// TIA Portal V17 export
// export: Created 2022-07-28T18:02:49.3810425Z, ExportSetting None, DisplayName Totally Integrated Automation Portal, DisplayVersion V17, DisplayName TIA Portal Openness, DisplayVersion V17, DisplayName TIA Portal Teamcenter Gateway, DisplayVersion V17, DisplayName TIA Portal Version Control Interface, DisplayVersion V17, DisplayName TIA Portal Test Suite Advanced, DisplayVersion V17, DisplayName SINAMICS Startdrive Advanced, DisplayVersion V17, DisplayName SINAMICS DCC, DisplayVersion V17, DisplayName SINAMICS Startdrive G130, G150, S120, S150, SINAMICS MV, S210, DisplayVersion V17, DisplayName SINAMICS Startdrive G110M, G120, G120C, G120D, G120P, G115D, DisplayVersion V17, DisplayName STEP 7 Professional, DisplayVersion V17, DisplayName SIMATIC Energy Suite, DisplayVersion V17, DisplayName STEP 7 CFC, DisplayVersion V17, DisplayName STEP 7 Safety, DisplayVersion V17, DisplayName WinCC Advanced / Unified PC, DisplayVersion V17, DisplayName SIMATIC Visualization Architect, DisplayVersion V17
FUNCTION "Lib_FC_PID_Cascad_SetNextFreeFull" : Void   // FC24, SCL
{ S7_Optimized_Access := 'TRUE' }
// stored: SetENOAutomatically false
   VAR_IN_OUT
      i_InputArr : "_PID_Cascad_AutoCtrlPumpsAll";
   END_VAR
   VAR_TEMP
      t_ExistFree : Bool;
      ti_Cnt : Int;
   END_VAR
BEGIN
   //Set next available element for PID and reset all unavailable
   //Reset flags
   #t_ExistFree := false;
   FOR #ti_Cnt := 0 TO 2 DO

       IF #i_InputArr.Arr[#ti_Cnt].AutoControl_P.StatusGen.StartFull
           AND ( NOT #i_InputArr.Arr[#ti_Cnt].Enabled
           OR NOT  #i_InputArr.Arr[#ti_Cnt].AutoControl_P.Mode.Auto
           OR NOT  #i_InputArr.Arr[#ti_Cnt].AutoControl_P.StatusGen.Ready)
       THEN
           #i_InputArr.Arr[#ti_Cnt].AutoControl_P.StatusGen.StartFull := false;
       END_IF;

       IF NOT #i_InputArr.Arr[#ti_Cnt].AutoControl_P.StatusGen.StartFull
           AND NOT #i_InputArr.Arr[#ti_Cnt].AutoControl_P.StatusGen.StartPID
           AND #i_InputArr.Arr[#ti_Cnt].Enabled
           AND #i_InputArr.Arr[#ti_Cnt].AutoControl_P.Mode.Auto
           AND #i_InputArr.Arr[#ti_Cnt].AutoControl_P.StatusGen.Ready
       THEN
           #i_InputArr.Arr[#ti_Cnt].AutoControl_P.StatusGen.StartFull := true;
           RETURN;
       END_IF;
   END_FOR;
END_FUNCTION
